{attribute 'qualified_only'}
{attribute 'strict'}
TYPE E_MaterialType :
(
	Undefined := 0,
	None,
	Upper
);
END_TYPE

(* stored: Version 1.1.0.1, ProductVersion 3.1.4024.5
   DUT E_MaterialType: Id {e38ecb34-183a-4c79-bb19-009b18578244} *)
